FUNCTION_BLOCK AXE_CMD
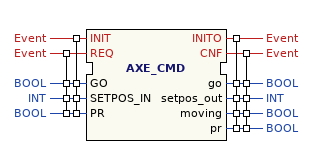
  EVENT_INPUT
    INIT WITH GO, SETPOS_IN, PR;
    REQ WITH GO, SETPOS_IN, PR;
  END_EVENT
  EVENT_OUTPUT
    INITO WITH go, setpos_out, moving, pr;
    CNF WITH go, setpos_out, moving, pr;
  END_EVENT
  VAR_INPUT
    GO : BOOL;
    SETPOS_IN : INT;
    PR : BOOL;
  END_VAR
  VAR_OUTPUT
    go : BOOL;
    setpos_out : INT;
    moving : BOOL;
    pr : BOOL;
  END_VAR
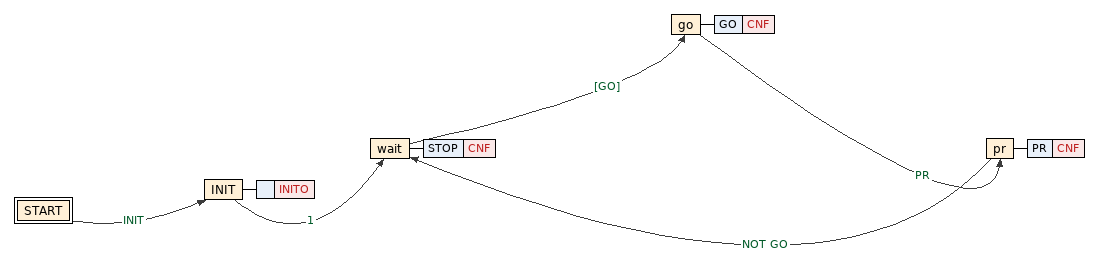
  EC_STATES
    START;
    wait : STOP -> CNF;
    go : GO -> CNF;
    pr : PR -> CNF;
    INIT : -> INITO;
  END_STATES
  EC_TRANSITIONS
    START TO INIT := INIT;
    wait TO go := [GO];
    go TO pr := PR;
    pr TO wait := NOT GO;
    INIT TO wait := 1;
  END_TRANSITIONS
  ALGORITHM INIT IN ST:
pr := FALSE;
moving := TRUE;
setpos_out := 1;
go := TRUE;
  END_ALGORITHM
  ALGORITHM GO IN ST:
go := TRUE;
setpos_out := SETPOS_IN;
moving := TRUE;
pr := FALSE;
  END_ALGORITHM
  ALGORITHM PR IN ST:
go := FALSE;
pr := TRUE;
moving := FALSE;
  END_ALGORITHM
  ALGORITHM STOP IN ST:
go := FALSE;
moving := FALSE;
pr := FALSE;
  END_ALGORITHM
END_FUNCTION_BLOCK
